(* Logix 5000 project; controller R1USB70001_CWRU_SOURCE_20111116 vendor 1 type 14 code 54 rev 19.11; software revision 19.01 *)

TASK MainTask (continuous, watchdog 500 ms) : MainProgram

MODULES
   Local : vendor 1 type 14 code 54 (ICP 2, rev 19.11)
      CNB_SOURCE : vendor 1 type 12 code 21 (ICP 0, rev 20.1)
         ACNR_SP_SC_N3 : vendor 1 type 12 code 111 (ControlNet 3, rev 1.83, Output RPI 8 ms)
            IE4C_SP_SC_S4 : 1734-IE4C (PointIO 4, rev 3.1, Input RPI 8 ms)
            IB8_SP_SC_S7 : 1734-IB8 (PointIO 7, rev 3.22)
            IE4C_SP_SC_S1 : 1734-IE4C (PointIO 1, rev 3.1, Input RPI 8 ms)
            IE4C_SP_SC_S2 : 1734-IE4C (PointIO 2, rev 3.1, Input RPI 8 ms)
            IE4C_SP_SC_S3 : 1734-IE4C (PointIO 3, rev 3.1, Input RPI 8 ms)
            IE4C_SP_SC_S5 : 1734-IE4C (PointIO 5, rev 3.1, Input RPI 8 ms)
            IB8_SP_SC_S8 : 1734-IB8 (PointIO 8, rev 3.22)
            IE4C_SP_SC_S6 : 1734-IE4C (PointIO 6, rev 3.1, Input RPI 8 ms)
            OB8_SP_SC_S9 : 1734-OB8 (PointIO 9, rev 3.22)
      EN2T_SOURCE : 1756-EN2T (ICP 1, Ethernet 10.88.0.103, rev 4.3)
END_MODULES

VAR_GLOBAL   (* controller tags *)
   AS_SP_L1_ACAM : ALIAS FOR ACNR_SP_SC_N3:1:I.Ch0Data;
   AS_SP_L1_ACVT : ALIAS FOR ACNR_SP_SC_N3:5:I.Ch0Data;
   AS_SP_L1_CS : ALIAS FOR ACNR_SP_SC_N3:9:O.0;
   AS_SP_L1_DCAM : ALIAS FOR ACNR_SP_SC_N3:1:I.Ch1Data;
   AS_SP_L1_DCVS : ALIAS FOR ACNR_SP_SC_N3:7:I.1;
   AS_SP_L2_ACAM : ALIAS FOR ACNR_SP_SC_N3:1:I.Ch2Data;
   AS_SP_L2_ACVT : ALIAS FOR ACNR_SP_SC_N3:5:I.Ch1Data;
   AS_SP_L2_CS : ALIAS FOR ACNR_SP_SC_N3:9:O.1;
   AS_SP_L2_DCAM : ALIAS FOR ACNR_SP_SC_N3:1:I.Ch3Data;
   AS_SP_L2_DCVS : ALIAS FOR ACNR_SP_SC_N3:7:I.3;
   Comment : DINT[2] := ([0] := 3);
   HMI_Intfc_Read_Buffer : DINT[32] := ([0] := -1, [1] := 1, [3] := 1, [5] := 2, [6] := -1, [8] := 1, [10] := -1, [11] := 1, [12] := -1, [15] := 1, [21] := 244, [22] := -15, [23] := -10, [25] := 288, [26] := 326, [27] := 327, [28] := 328, [29] := 329, [30] := 330, [31] := 331);
        [0]   // AS_SP_L1_ACAM
        [1]   // AS_SP_L1_DCAM
        [2]   // AS_SP_L2_ACAM
        [3]   // AS_SP_L2_DCAM
        [4]   // WF_SP_LN_ACAM
        [5]   // WF_SP_LN_DCAM1
        [6]   // WF_SP_LN_DCAM2
        [7]   // WT_SP_LN_ACAM
        [8]   // WT_SP_LN_DCAM1
        [9]   // WT_SP_LN_DCAM2
        [10]   // SF_SP_LN_ACAM
        [11]   // SF_SP_LN_DCAM1
        [12]   // SF_SP_LN_DCAM2
        [13]   // SC_SP_LN_ACAM
        [14]   // SC_SP_LN_DCAM1
        [15]   // SC_SP_LN_DCAM2
        [16]   // AS_SP_L1_ACVT
        [17]   // AS_SP_L2_ACVT
        [18]   // WF_SP_LN_ACVT
        [19]   // WT_SP_LN_ACVT
        [20]   // SF_SP_LN_ACVT
        [21]   // SC_SP_LN_ACVT
        [24].1   // AS_SP_L1_DCVS
        [24].3   // AS_SP_L2_DCVS
        [24].6   // WF_SP_LN_DCVS2
        [24].5   // WF_SP_LN_DCVS1
        [24].8   // WT_SP_LN_DCVS1
        [24].9   // WT_SP_LN_DCVS2
        [24].11   // SF_SP_LN_DCVS1
        [24].12   // SF_SP_LN_DCVS2
        [24].14   // SC_SP_LN_DCVS1
        [24].15   // SC_SP_LN_DCVS2
        [25].0   // AS_SP_L1_CS
        [25].1   // AS_SP_L2_CS
        [25].2   // WF_SP_LN_CS
        [25].3   // WT_SP_LN_CS
        [25].4   // SF_SP_LN_CS
        [25].5   // SC_SP_LN_CS
        [22]   // SPARE RESERVED FOR SLOT 6 CHANNEL 2
        [23]   // SPARE RESERVED FOR SLOT 6 CHANNEL 3
   SC_SP_LN_ACAM : ALIAS FOR ACNR_SP_SC_N3:4:I.Ch1Data;
   SC_SP_LN_ACVT : ALIAS FOR ACNR_SP_SC_N3:6:I.Ch1Data;
   SC_SP_LN_CS : ALIAS FOR ACNR_SP_SC_N3:9:O.5;
   SC_SP_LN_DCAM1 : ALIAS FOR ACNR_SP_SC_N3:4:I.Ch2Data;
   SC_SP_LN_DCAM2 : ALIAS FOR ACNR_SP_SC_N3:4:I.Ch3Data;
   SC_SP_LN_DCVS1 : ALIAS FOR ACNR_SP_SC_N3:8:I.6;
   SC_SP_LN_DCVS2 : ALIAS FOR ACNR_SP_SC_N3:8:I.7;
   SF_SP_LN_ACAM : ALIAS FOR ACNR_SP_SC_N3:3:I.Ch2Data;
   SF_SP_LN_ACVT : ALIAS FOR ACNR_SP_SC_N3:6:I.Ch0Data;
   SF_SP_LN_CS : ALIAS FOR ACNR_SP_SC_N3:9:O.4;
   SF_SP_LN_DCAM1 : ALIAS FOR ACNR_SP_SC_N3:3:I.Ch3Data;
   SF_SP_LN_DCAM2 : ALIAS FOR ACNR_SP_SC_N3:4:I.Ch0Data;
   SF_SP_LN_DCVS1 : ALIAS FOR ACNR_SP_SC_N3:8:I.3;
   SF_SP_LN_DCVS2 : ALIAS FOR ACNR_SP_SC_N3:8:I.4;
   SOURCE1_USER : BOOL;
   SOURCE3_USER : BOOL;
   SOURCE_1_Alias : BOOL;
   SOURCE_2_Alias : BOOL;
   SOURCE_3_Alias : BOOL;
   SOURCE_3_CONTROL_TIMER : BOOL;
   SOURCE_4_Alias : BOOL;
   WF_SP_LN_ACAM : ALIAS FOR ACNR_SP_SC_N3:2:I.Ch0Data;
   WF_SP_LN_ACVT : ALIAS FOR ACNR_SP_SC_N3:5:I.Ch2Data;
   WF_SP_LN_CS : ALIAS FOR ACNR_SP_SC_N3:9:O.2;
   WF_SP_LN_DCAM1 : ALIAS FOR ACNR_SP_SC_N3:2:I.Ch1Data;
   WF_SP_LN_DCAM2 : ALIAS FOR ACNR_SP_SC_N3:2:I.Ch2Data;
   WF_SP_LN_DCVS1 : ALIAS FOR ACNR_SP_SC_N3:7:I.5;
   WF_SP_LN_DCVS2 : ALIAS FOR ACNR_SP_SC_N3:7:I.6;
   WT_SP_LN_ACAM : ALIAS FOR ACNR_SP_SC_N3:2:I.Ch3Data;
   WT_SP_LN_ACVT : ALIAS FOR ACNR_SP_SC_N3:5:I.Ch3Data;
   WT_SP_LN_CS : ALIAS FOR ACNR_SP_SC_N3:9:O.3;
   WT_SP_LN_DCAM1 : ALIAS FOR ACNR_SP_SC_N3:3:I.Ch0Data;
   WT_SP_LN_DCAM2 : ALIAS FOR ACNR_SP_SC_N3:3:I.Ch1Data;
   WT_SP_LN_DCVS1 : ALIAS FOR ACNR_SP_SC_N3:8:I.0;
   WT_SP_LN_DCVS2 : ALIAS FOR ACNR_SP_SC_N3:8:I.1;
END_VAR

PROGRAM MainProgram   (* main routine MainRoutine *)
VAR
   CURRENT_SCALE_HIGH : REAL := 0.00061037;
   DC_CURRENT : REAL;
   MAINS1_AC_CURRENT : REAL;
   MAINS2_AC_CURRENT : REAL;
   MAINS2_DC_CURRENT : REAL;
   SC_AC_CURRENT : REAL;
   SC_AC_CURRENT_RAW : REAL;
   SC_AC_VOLTAGE : REAL;
   SC_AC_VOLTAGE_RAW : REAL;
   SC_DC_REG_CURRENT : REAL;
   SC_DC_REG_CURRENT_RAW : REAL;
   SC_DC_UNREG_CURRENT : REAL;
   SC_DC_UNREG_CURRENT_RAW : REAL;
   SC_REG_DC_VOLTAGE : BOOL;
   SC_REG_DC_VOLTAGE_RAW : BOOL;
   SC_UNREG_DC_VOLTAGE : BOOL;
   SC_UNREG_DC_VOLTAGE_RAW : BOOL;
   SF_AC_CURRENT : REAL;
   SF_AC_CURRENT_RAW : REAL;
   SF_AC_VOLTAGE : REAL;
   SF_AC_VOLTAGE_RAW : REAL;
   SF_AVAILABLE_THRESHOLD : REAL;
   SF_CLOSE_PROXY : BOOL;
   SF_COMMAND_CHANGED : BOOL;
   SF_COMMAND_CHANGED_TIMER : TIMER := (PRE := 2000);
   SF_CONNECTED : BOOL;
   SF_DC_REG_CURRENT : REAL;
   SF_DC_REG_CURRENT_RAW : REAL;
   SF_DC_UNREG_CURRENT : REAL;
   SF_DC_UNREG_CURRENT_RAW : REAL;
   SF_DISCONNECTED : BOOL;
   SF_INT_REQ_CLOSE : BOOL;
   SF_INT_REQ_CONNECT : BOOL;
   SF_MAX_CURRENT : REAL;
   SF_POWER_AVAILABLE : BOOL;
   SF_REG_DC_VOLTAGE : BOOL;
   SF_REG_DC_VOLTAGE_RAW : BOOL;
   SF_REQ_CLOSE : BOOL;
   SF_REQ_CONNECT : BOOL;
   SF_REQ_DISCONNECT : BOOL;
   SF_REQ_OPEN : BOOL;
   SF_UNREG_DC_VOLTAGE : BOOL;
   VOLTAGE_SCALE : REAL := 0.000732444;
   WF_AC_CURRENT : REAL;
   WF_AC_CURRENT_RAW : REAL;
   WF_AC_VOLTAGE : REAL;
   WF_AC_VOLTAGE_RAW : REAL;
   WF_DC_REG_CURRENT : REAL;
   WF_DC_REG_CURRENT_RAW : REAL;
   WF_DC_UNREG_CURRENT : REAL;
   WF_DC_UNREG_CURRENT_RAW : REAL;
   WF_REG_DC_VOLTAGE : BOOL;
   WF_REG_DC_VOLTAGE_RAW : BOOL;
   WF_UNREG_DC_VOLTAGE : BOOL;
   WF_UNREG_DC_VOLTAGE_RAW : BOOL;
   WT_AC_CURRENT : REAL;
   WT_AC_CURRENT_RAW : REAL;
   WT_AC_VOLTAGE : REAL;
   WT_AC_VOLTAGE_RAW : REAL;
   WT_DC_REG_CURRENT : REAL;
   WT_DC_REG_CURRENT_RAW : REAL;
   WT_DC_UNREG_CURRENT : REAL;
   WT_DC_UNREG_CURRENT_RAW : REAL;
   WT_REG_DC_VOLTAGE : BOOL;
   WT_UNREG_DC_VOLTAGE : BOOL;
END_VAR

ROUTINE IMPORT_DATA   (* ladder *)
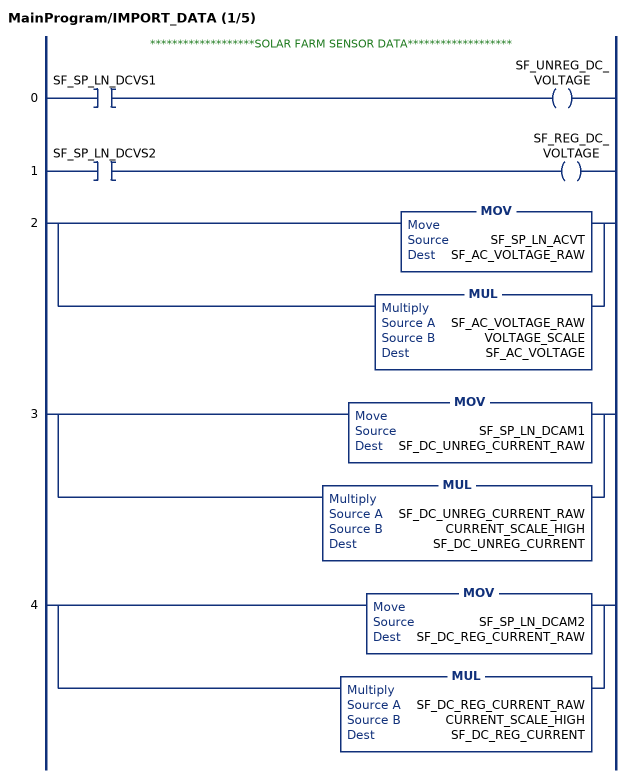
   // *******************SOLAR FARM SENSOR DATA*******************
   0: XIC(SF_SP_LN_DCVS1)OTE(SF_UNREG_DC_VOLTAGE);
   1: XIC(SF_SP_LN_DCVS2)OTE(SF_REG_DC_VOLTAGE);
   2: [MOV(SF_SP_LN_ACVT,SF_AC_VOLTAGE_RAW) ,MUL(SF_AC_VOLTAGE_RAW,VOLTAGE_SCALE,SF_AC_VOLTAGE) ];
   3: [MOV(SF_SP_LN_DCAM1,SF_DC_UNREG_CURRENT_RAW) ,MUL(SF_DC_UNREG_CURRENT_RAW,CURRENT_SCALE_HIGH,SF_DC_UNREG_CURRENT) ];
   4: [MOV(SF_SP_LN_DCAM2,SF_DC_REG_CURRENT_RAW) ,MUL(SF_DC_REG_CURRENT_RAW,CURRENT_SCALE_HIGH,SF_DC_REG_CURRENT) ];
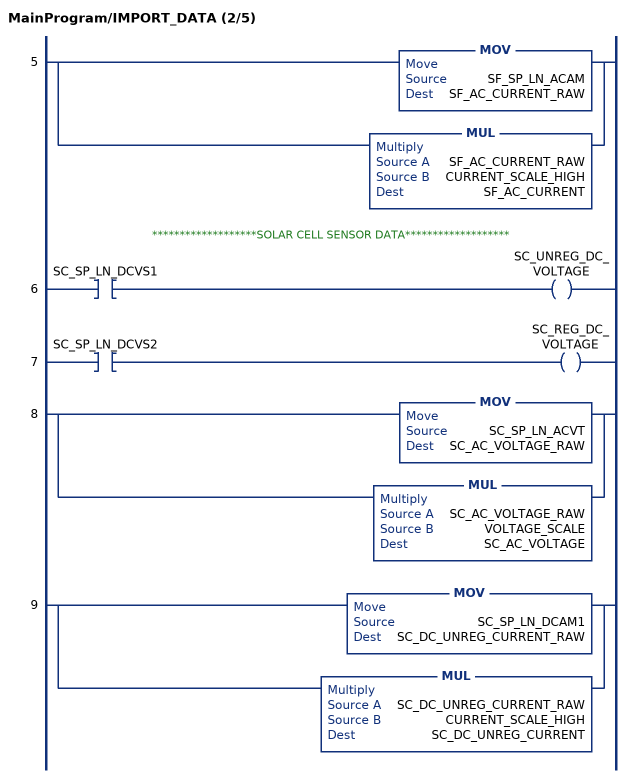
   5: [MOV(SF_SP_LN_ACAM,SF_AC_CURRENT_RAW) ,MUL(SF_AC_CURRENT_RAW,CURRENT_SCALE_HIGH,SF_AC_CURRENT) ];
   // *******************SOLAR CELL SENSOR DATA*******************
   6: XIC(SC_SP_LN_DCVS1)OTE(SC_UNREG_DC_VOLTAGE);
   7: XIC(SC_SP_LN_DCVS2)OTE(SC_REG_DC_VOLTAGE);
   8: [MOV(SC_SP_LN_ACVT,SC_AC_VOLTAGE_RAW) ,MUL(SC_AC_VOLTAGE_RAW,VOLTAGE_SCALE,SC_AC_VOLTAGE) ];
   9: [MOV(SC_SP_LN_DCAM1,SC_DC_UNREG_CURRENT_RAW) ,MUL(SC_DC_UNREG_CURRENT_RAW,CURRENT_SCALE_HIGH,SC_DC_UNREG_CURRENT) ];
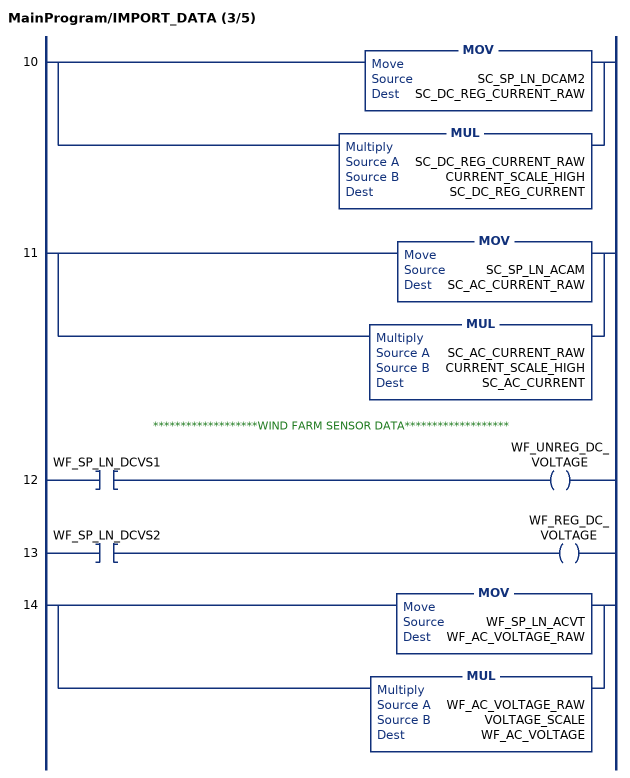
   10: [MOV(SC_SP_LN_DCAM2,SC_DC_REG_CURRENT_RAW) ,MUL(SC_DC_REG_CURRENT_RAW,CURRENT_SCALE_HIGH,SC_DC_REG_CURRENT) ];
   11: [MOV(SC_SP_LN_ACAM,SC_AC_CURRENT_RAW) ,MUL(SC_AC_CURRENT_RAW,CURRENT_SCALE_HIGH,SC_AC_CURRENT) ];
   // *******************WIND FARM SENSOR DATA*******************
   12: XIC(WF_SP_LN_DCVS1)OTE(WF_UNREG_DC_VOLTAGE);
   13: XIC(WF_SP_LN_DCVS2)OTE(WF_REG_DC_VOLTAGE);
   14: [MOV(WF_SP_LN_ACVT,WF_AC_VOLTAGE_RAW) ,MUL(WF_AC_VOLTAGE_RAW,VOLTAGE_SCALE,WF_AC_VOLTAGE) ];
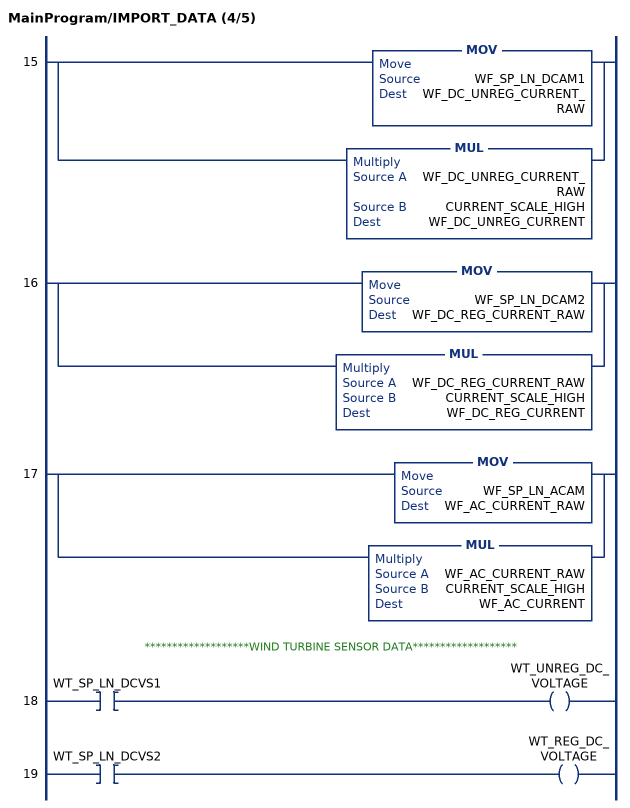
   15: [MOV(WF_SP_LN_DCAM1,WF_DC_UNREG_CURRENT_RAW) ,MUL(WF_DC_UNREG_CURRENT_RAW,CURRENT_SCALE_HIGH,WF_DC_UNREG_CURRENT) ];
   16: [MOV(WF_SP_LN_DCAM2,WF_DC_REG_CURRENT_RAW) ,MUL(WF_DC_REG_CURRENT_RAW,CURRENT_SCALE_HIGH,WF_DC_REG_CURRENT) ];
   17: [MOV(WF_SP_LN_ACAM,WF_AC_CURRENT_RAW) ,MUL(WF_AC_CURRENT_RAW,CURRENT_SCALE_HIGH,WF_AC_CURRENT) ];
   // *******************WIND TURBINE SENSOR DATA*******************
   18: XIC(WT_SP_LN_DCVS1)OTE(WT_UNREG_DC_VOLTAGE);
   19: XIC(WT_SP_LN_DCVS2)OTE(WT_REG_DC_VOLTAGE);
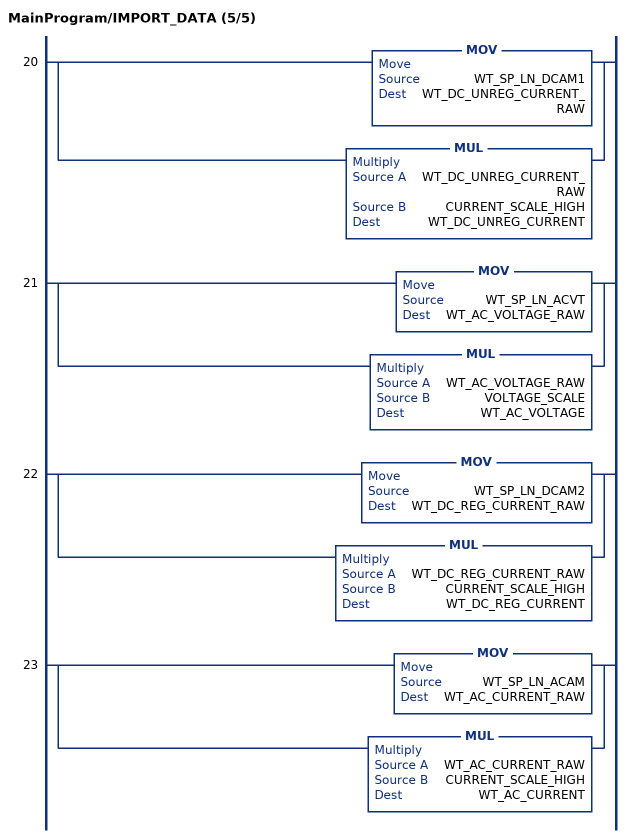
   20: [MOV(WT_SP_LN_DCAM1,WT_DC_UNREG_CURRENT_RAW) ,MUL(WT_DC_UNREG_CURRENT_RAW,CURRENT_SCALE_HIGH,WT_DC_UNREG_CURRENT) ];
   21: [MOV(WT_SP_LN_ACVT,WT_AC_VOLTAGE_RAW) ,MUL(WT_AC_VOLTAGE_RAW,VOLTAGE_SCALE,WT_AC_VOLTAGE) ];
   22: [MOV(WT_SP_LN_DCAM2,WT_DC_REG_CURRENT_RAW) ,MUL(WT_DC_REG_CURRENT_RAW,CURRENT_SCALE_HIGH,WT_DC_REG_CURRENT) ];
   23: [MOV(WT_SP_LN_ACAM,WT_AC_CURRENT_RAW) ,MUL(WT_AC_CURRENT_RAW,CURRENT_SCALE_HIGH,WT_AC_CURRENT) ];
END_ROUTINE

ROUTINE MainRoutine   (* ladder *)
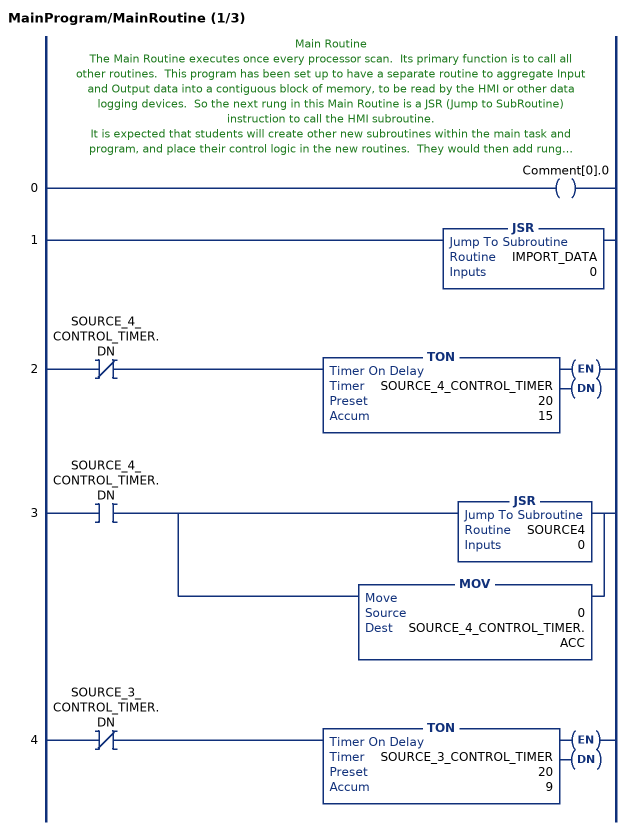
   // Main Routine
   // The Main Routine executes once every processor scan.  Its primary function is to call all other routines.  This program has been set up to have a separate routine to aggregate Input and Output data into a contiguous block of memory, to be read by the HMI or other data logging devices.  So the next rung in this Main Routine is a JSR (Jump to SubRoutine) instruction to call the HMI subroutine.
   // It is expected that students will create other new subroutines within the main task and program, and place their control logic in the new routines.  They would then add rungs within this Main Routine to call the new subroutines that contain their logic.
   0: OTE(Comment[0].0);
   1: JSR(IMPORT_DATA,0);
   2: XIO(SOURCE_4_CONTROL_TIMER.DN)TON(SOURCE_4_CONTROL_TIMER,20,15);
   3: XIC(SOURCE_4_CONTROL_TIMER.DN)[JSR(SOURCE4,0) ,MOV(0,SOURCE_4_CONTROL_TIMER.ACC) ];
   4: XIO(SOURCE_3_CONTROL_TIMER.DN)TON(SOURCE_3_CONTROL_TIMER,20,9);
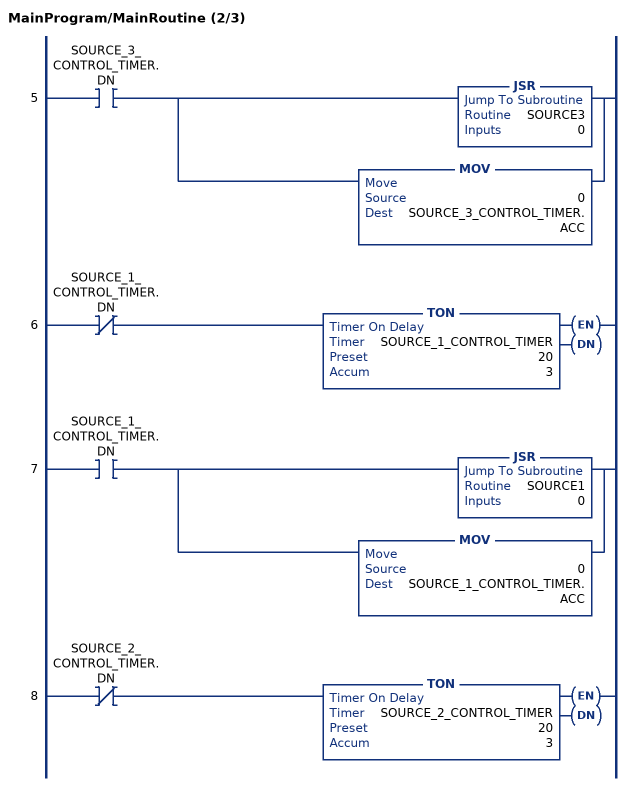
   5: XIC(SOURCE_3_CONTROL_TIMER.DN)[JSR(SOURCE3,0) ,MOV(0,SOURCE_3_CONTROL_TIMER.ACC) ];
   6: XIO(SOURCE_1_CONTROL_TIMER.DN)TON(SOURCE_1_CONTROL_TIMER,20,3);
   7: XIC(SOURCE_1_CONTROL_TIMER.DN)[JSR(SOURCE1,0) ,MOV(0,SOURCE_1_CONTROL_TIMER.ACC) ];
   8: XIO(SOURCE_2_CONTROL_TIMER.DN)TON(SOURCE_2_CONTROL_TIMER,20,3);
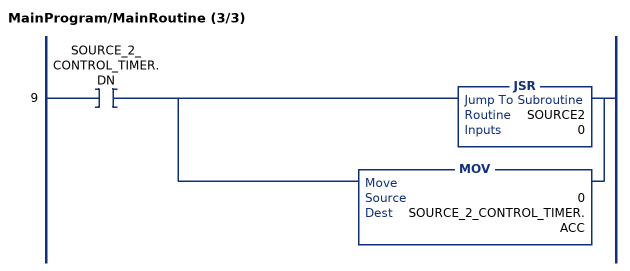
   9: XIC(SOURCE_2_CONTROL_TIMER.DN)[JSR(SOURCE2,0) ,MOV(0,SOURCE_2_CONTROL_TIMER.ACC) ];
END_ROUTINE

ROUTINE SF_MANAGEMENT   (* ladder *)
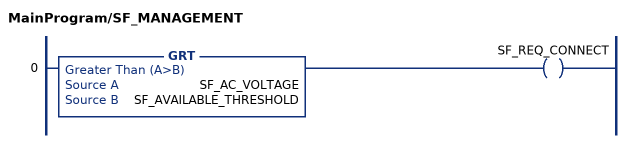
   0: GRT(SF_AC_VOLTAGE,SF_AVAILABLE_THRESHOLD)OTE(SF_REQ_CONNECT);
END_ROUTINE

ROUTINE SOURCE3   (* ladder *)
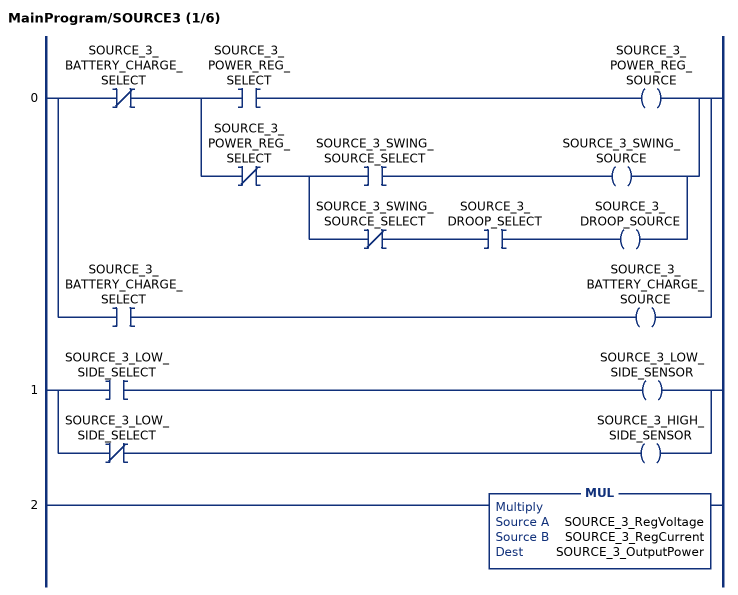
   0: [XIO(SOURCE_3_BATTERY_CHARGE_SELECT) [XIC(SOURCE_3_POWER_REG_SELECT) OTE(SOURCE_3_POWER_REG_SOURCE) ,XIO(SOURCE_3_POWER_REG_SELECT) [XIC(SOURCE_3_SWING_SOURCE_SELECT) OTE(SOURCE_3_SWING_SOURCE) ,XIO(SOURCE_3_SWING_SOURCE_SELECT) XIC(SOURCE_3_DROOP_SELECT) OTE(SOURCE_3_DROOP_SOURCE) ] ] ,XIC(SOURCE_3_BATTERY_CHARGE_SELECT) OTE(SOURCE_3_BATTERY_CHARGE_SOURCE) ];
   1: [XIC(SOURCE_3_LOW_SIDE_SELECT) OTE(SOURCE_3_LOW_SIDE_SENSOR) ,XIO(SOURCE_3_LOW_SIDE_SELECT) OTE(SOURCE_3_HIGH_SIDE_SENSOR) ];
   2: MUL(SOURCE_3_RegVoltage,SOURCE_3_RegCurrent,SOURCE_3_OutputPower);
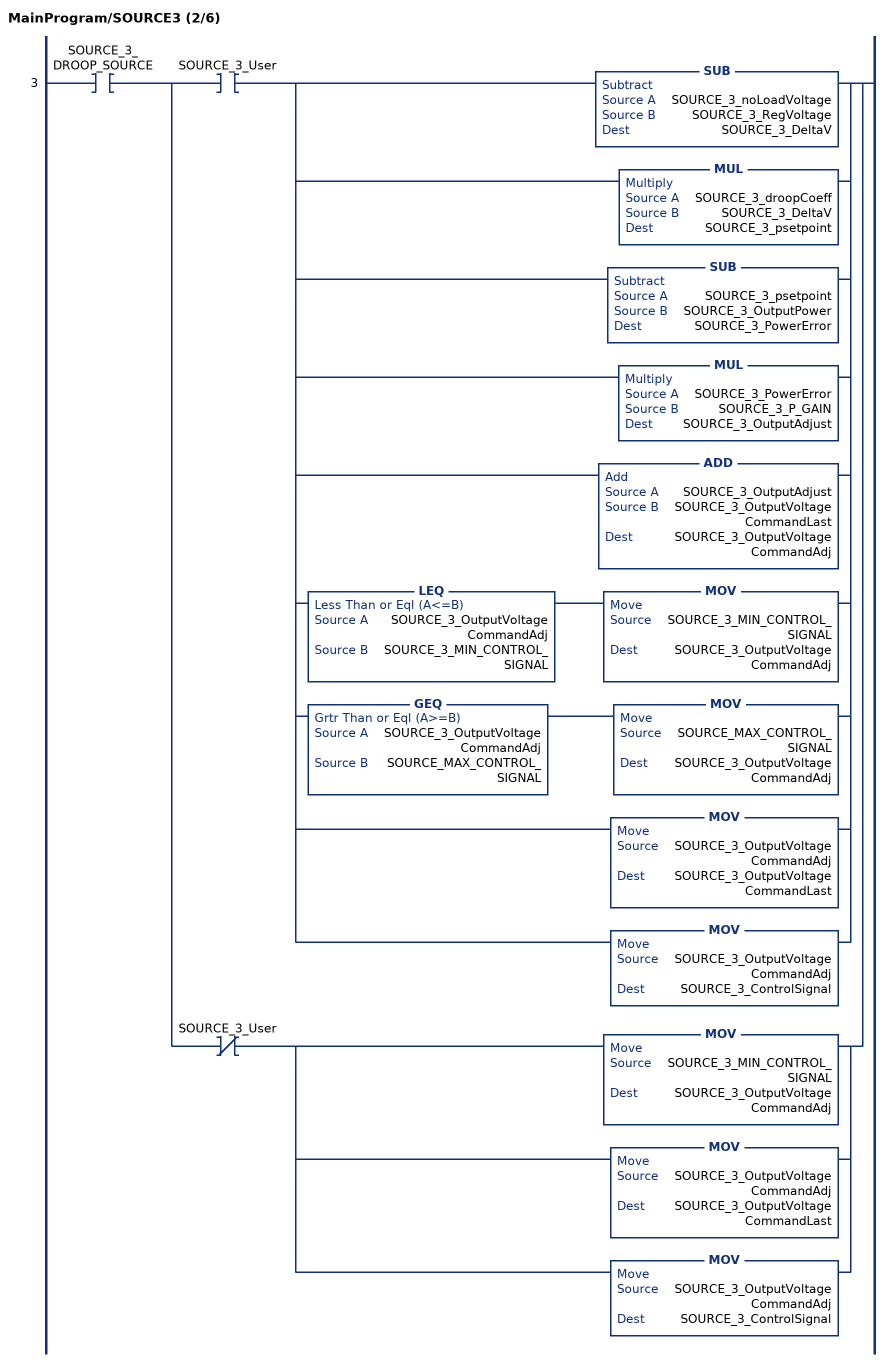
   3: XIC(SOURCE_3_DROOP_SOURCE)[XIC(SOURCE_3_User) [SUB(SOURCE_3_noLoadVoltage,SOURCE_3_RegVoltage,SOURCE_3_DeltaV) ,MUL(SOURCE_3_droopCoeff,SOURCE_3_DeltaV,SOURCE_3_psetpoint) ,SUB(SOURCE_3_psetpoint,SOURCE_3_OutputPower,SOURCE_3_PowerError) ,MUL(SOURCE_3_PowerError,SOURCE_3_P_GAIN,SOURCE_3_OutputAdjust) ,ADD(SOURCE_3_OutputAdjust,SOURCE_3_OutputVoltageCommandLast,SOURCE_3_OutputVoltageCommandAdj) ,LEQ(SOURCE_3_OutputVoltageCommandAdj,SOURCE_3_MIN_CONTROL_SIGNAL) MOV(SOURCE_3_MIN_CONTROL_SIGNAL,SOURCE_3_OutputVoltageCommandAdj) ,GEQ(SOURCE_3_OutputVoltageCommandAdj,SOURCE_MAX_CONTROL_SIGNAL) MOV(SOURCE_MAX_CONTROL_SIGNAL,SOURCE_3_OutputVoltageCommandAdj) ,MOV(SOURCE_3_OutputVoltageCommandAdj,SOURCE_3_OutputVoltageCommandLast) ,MOV(SOURCE_3_OutputVoltageCommandAdj,SOURCE_3_ControlSignal) ] ,XIO(SOURCE_3_User) [MOV(SOURCE_3_MIN_CONTROL_SIGNAL,SOURCE_3_OutputVoltageCommandAdj) ,MOV(SOURCE_3_OutputVoltageCommandAdj,SOURCE_3_OutputVoltageCommandLast) ,MOV(SOURCE_3_OutputVoltageCommandAdj,SOURCE_3_ControlSignal) ] ];
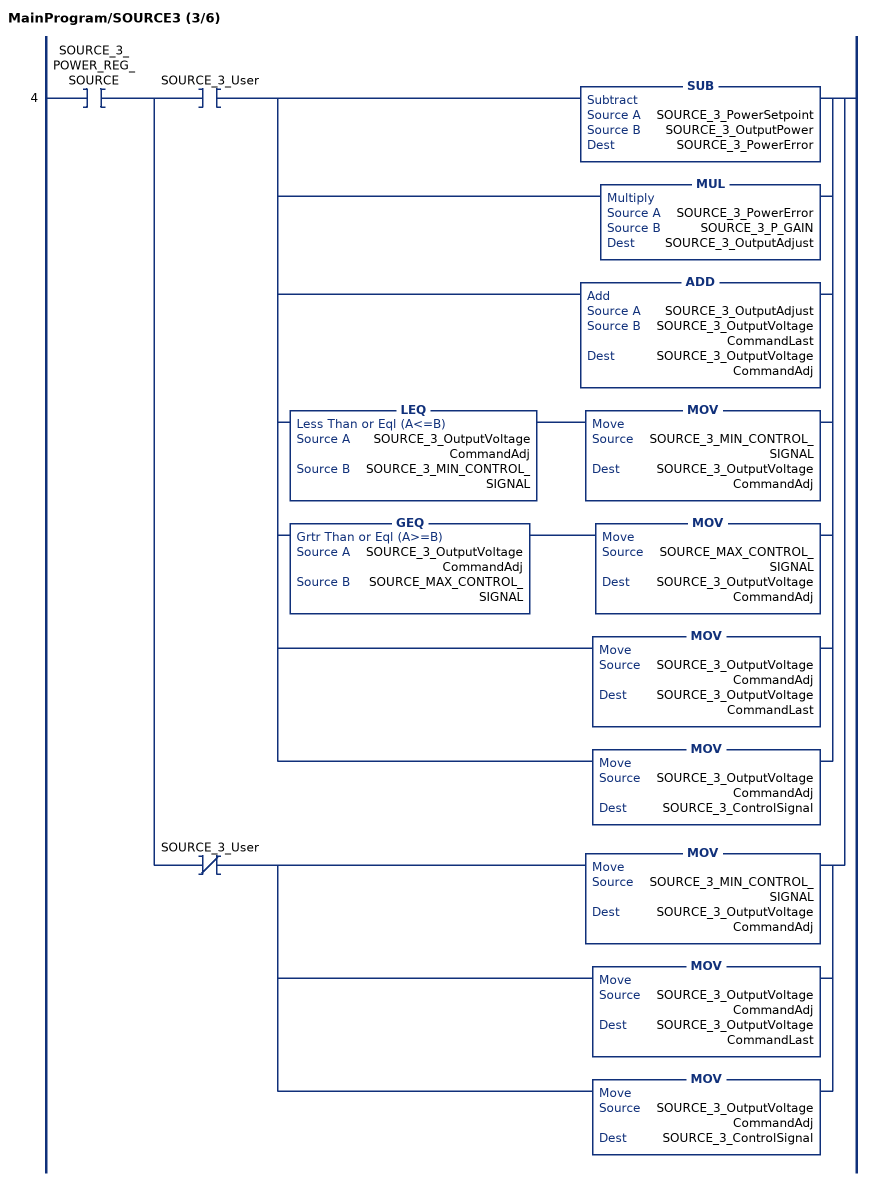
   4: XIC(SOURCE_3_POWER_REG_SOURCE)[XIC(SOURCE_3_User) [SUB(SOURCE_3_PowerSetpoint,SOURCE_3_OutputPower,SOURCE_3_PowerError) ,MUL(SOURCE_3_PowerError,SOURCE_3_P_GAIN,SOURCE_3_OutputAdjust) ,ADD(SOURCE_3_OutputAdjust,SOURCE_3_OutputVoltageCommandLast,SOURCE_3_OutputVoltageCommandAdj) ,LEQ(SOURCE_3_OutputVoltageCommandAdj,SOURCE_3_MIN_CONTROL_SIGNAL) MOV(SOURCE_3_MIN_CONTROL_SIGNAL,SOURCE_3_OutputVoltageCommandAdj) ,GEQ(SOURCE_3_OutputVoltageCommandAdj,SOURCE_MAX_CONTROL_SIGNAL) MOV(SOURCE_MAX_CONTROL_SIGNAL,SOURCE_3_OutputVoltageCommandAdj) ,MOV(SOURCE_3_OutputVoltageCommandAdj,SOURCE_3_OutputVoltageCommandLast) ,MOV(SOURCE_3_OutputVoltageCommandAdj,SOURCE_3_ControlSignal) ] ,XIO(SOURCE_3_User) [MOV(SOURCE_3_MIN_CONTROL_SIGNAL,SOURCE_3_OutputVoltageCommandAdj) ,MOV(SOURCE_3_OutputVoltageCommandAdj,SOURCE_3_OutputVoltageCommandLast) ,MOV(SOURCE_3_OutputVoltageCommandAdj,SOURCE_3_ControlSignal) ] ];
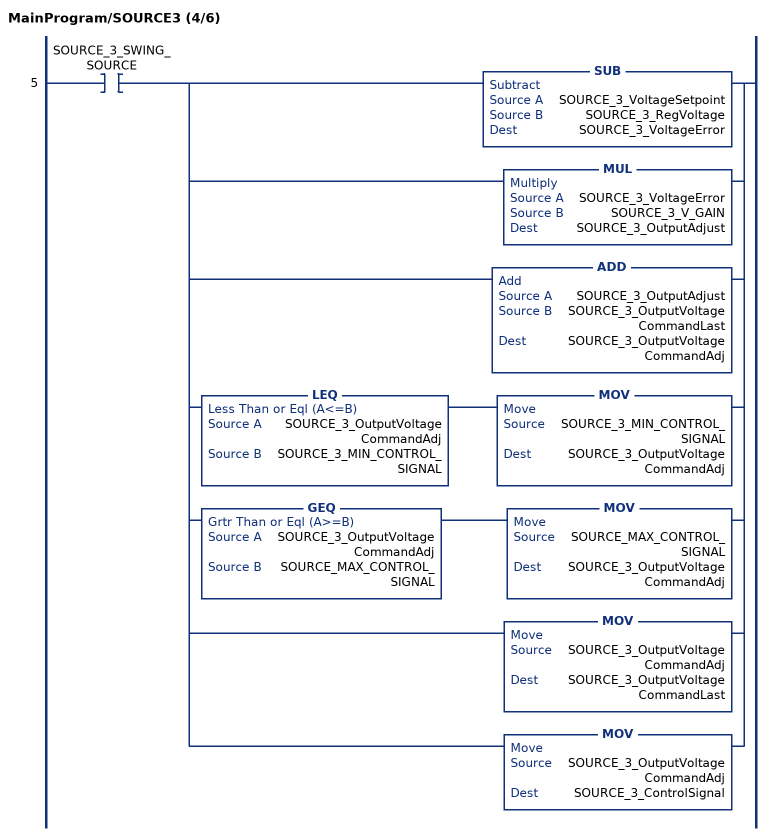
   5: XIC(SOURCE_3_SWING_SOURCE)[SUB(SOURCE_3_VoltageSetpoint,SOURCE_3_RegVoltage,SOURCE_3_VoltageError) ,MUL(SOURCE_3_VoltageError,SOURCE_3_V_GAIN,SOURCE_3_OutputAdjust) ,ADD(SOURCE_3_OutputAdjust,SOURCE_3_OutputVoltageCommandLast,SOURCE_3_OutputVoltageCommandAdj) ,LEQ(SOURCE_3_OutputVoltageCommandAdj,SOURCE_3_MIN_CONTROL_SIGNAL) MOV(SOURCE_3_MIN_CONTROL_SIGNAL,SOURCE_3_OutputVoltageCommandAdj) ,GEQ(SOURCE_3_OutputVoltageCommandAdj,SOURCE_MAX_CONTROL_SIGNAL) MOV(SOURCE_MAX_CONTROL_SIGNAL,SOURCE_3_OutputVoltageCommandAdj) ,MOV(SOURCE_3_OutputVoltageCommandAdj,SOURCE_3_OutputVoltageCommandLast) ,MOV(SOURCE_3_OutputVoltageCommandAdj,SOURCE_3_ControlSignal) ];
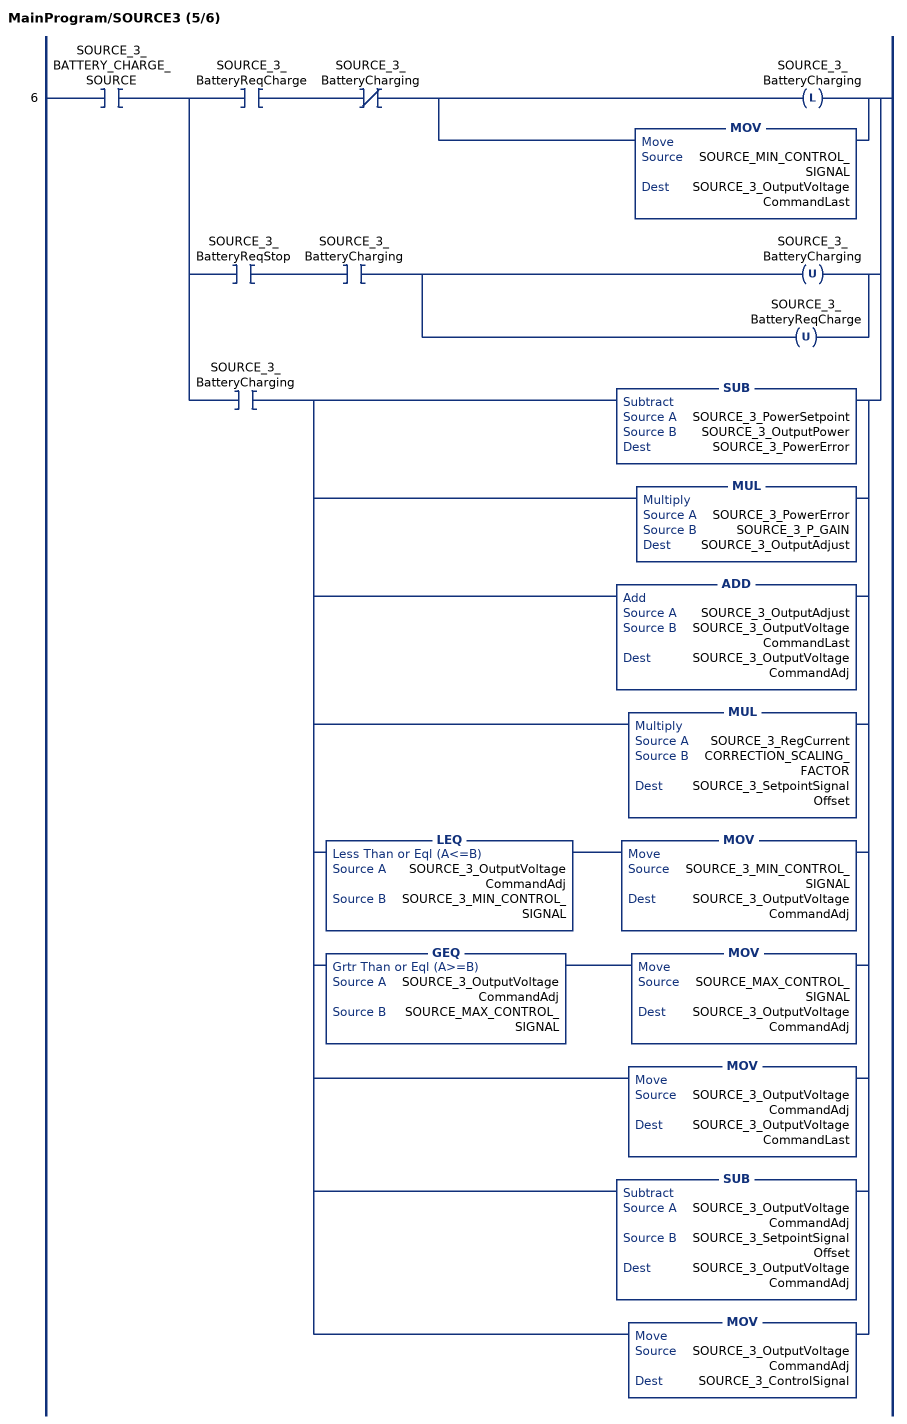
   6: XIC(SOURCE_3_BATTERY_CHARGE_SOURCE)[XIC(SOURCE_3_BatteryReqCharge) XIO(SOURCE_3_BatteryCharging) [OTL(SOURCE_3_BatteryCharging) ,MOV(SOURCE_MIN_CONTROL_SIGNAL,SOURCE_3_OutputVoltageCommandLast) ] ,XIC(SOURCE_3_BatteryReqStop) XIC(SOURCE_3_BatteryCharging) [OTU(SOURCE_3_BatteryCharging) ,OTU(SOURCE_3_BatteryReqCharge) ] ,XIC(SOURCE_3_BatteryCharging) [SUB(SOURCE_3_PowerSetpoint,SOURCE_3_OutputPower,SOURCE_3_PowerError) ,MUL(SOURCE_3_PowerError,SOURCE_3_P_GAIN,SOURCE_3_OutputAdjust) ,ADD(SOURCE_3_OutputAdjust,SOURCE_3_OutputVoltageCommandLast,SOURCE_3_OutputVoltageCommandAdj) ,MUL(SOURCE_3_RegCurrent,CORRECTION_SCALING_FACTOR,SOURCE_3_SetpointSignalOffset) ,LEQ(SOURCE_3_OutputVoltageCommandAdj,SOURCE_3_MIN_CONTROL_SIGNAL) MOV(SOURCE_3_MIN_CONTROL_SIGNAL,SOURCE_3_OutputVoltageCommandAdj) ,GEQ(SOURCE_3_OutputVoltageCommandAdj,SOURCE_MAX_CONTROL_SIGNAL) MOV(SOURCE_MAX_CONTROL_SIGNAL,SOURCE_3_OutputVoltageCommandAdj) ,MOV(SOURCE_3_OutputVoltageCommandAdj,SOURCE_3_OutputVoltageCommandLast) ,SUB(SOURCE_3_OutputVoltageCommandAdj,SOURCE_3_SetpointSignalOffset,SOURCE_3_OutputVoltageCommandAdj) ,MOV(SOURCE_3_OutputVoltageCommandAdj,SOURCE_3_ControlSignal) ] ];
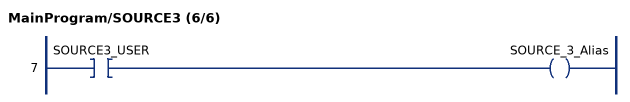
   7: XIC(SOURCE3_USER)OTE(SOURCE_3_Alias);
END_ROUTINE
END_PROGRAM
